INTERFACE I_IlluminationController_Base EXTENDS I_CH_Object, I_IlluminationController_StatusOnly, __SYSTEM.IQueryInterface

{attribute 'monitoring' := 'call'}
PROPERTY Busy : BOOL
GET
END_GET
END_PROPERTY

{attribute 'monitoring' := 'call'}
PROPERTY NextPossibleTriggerTime : T_DCTIME64
GET
END_GET
END_PROPERTY

{attribute 'monitoring' := 'call'}
PROPERTY Operational : BOOL
GET
END_GET
END_PROPERTY

METHOD Reset : HRESULT
END_METHOD

METHOD SetParent
VAR_INPUT
	ipVisionSystem  : I_VisionSystem;
END_VAR
END_METHOD

{attribute 'monitoring' := 'call'}
PROPERTY PUBLIC State : E_StateTerminal
GET
END_GET
END_PROPERTY

END_INTERFACE

(* stored: Version 1.1.0.1, ProductVersion 3.1.4024.12
   Itf I_IlluminationController_Base: Id {d81d1679-f7b1-4d60-ade1-2610f4ffd636}
   Property Busy: Id {0c8ccaad-c193-4a7a-a8ae-008a27a9c59d}
   Get Get: Id {103fc950-f95f-400a-be21-26d391dfc818}
   Property NextPossibleTriggerTime: Id {fbe68201-3519-42fd-932d-5997a5579930}
   Get Get: Id {64995085-47d9-49ac-880a-713c61029100}
   Property Operational: Id {20353367-f0f9-4ca7-86ad-67474f91ae65}
   Get Get: Id {7457f0b0-a53b-4345-9f37-d0407b0cf338}
   Method Reset: Id {c114186d-656d-4307-b0bb-a8b3843dfdee}
   Method SetParent: Id {5bdc47a1-13d6-48de-8cb5-0376c094c558}
   Property State: Id {4efee45b-b585-444c-917e-2f333d5436fc}
   Get Get: Id {a967bda0-047d-4694-9569-070be9284fae} *)
